{attribute addProperty BoxType "EL6201-0000-0017"}
{attribute addProperty Id "Slave_15A_DI0BIT10.125113Slave_15A_DI1BIT10.125114Slave_15A_DI2BIT10.125115Slave_15A_DI3BIT10.125116Slave_15B_DI0BIT10.125117Slave_15B_DI1BIT10.125118Slave_15B_DI2BIT10.125119Slave_15B_DI3BIT10.125120"}
{attribute addProperty CRC "3080739669"}
{attribute addProperty SizeInBites "8"}
{attribute addProperty SizeInBytes "1"}
TYPE Slave_15_Inputs_B7A05B55 :
STRUCT
	{attribute addProperty Name "Slave_15A_DI0"}
	Slave_15A_DI0 : BIT;
	{attribute addProperty Name "Slave_15A_DI1"}
	Slave_15A_DI1 : BIT;
	{attribute addProperty Name "Slave_15A_DI2"}
	Slave_15A_DI2 : BIT;
	{attribute addProperty Name "Slave_15A_DI3"}
	Slave_15A_DI3 : BIT;
	{attribute addProperty Name "Slave_15B_DI0"}
	Slave_15B_DI0 : BIT;
	{attribute addProperty Name "Slave_15B_DI1"}
	Slave_15B_DI1 : BIT;
	{attribute addProperty Name "Slave_15B_DI2"}
	Slave_15B_DI2 : BIT;
	{attribute addProperty Name "Slave_15B_DI3"}
	Slave_15B_DI3 : BIT;
END_STRUCT
END_TYPE

(* stored: Version 1.2.0.0, ProductVersion 3.1.4024.9
   DUT Slave_15_Inputs_B7A05B55: Id {9046cdec-39e5-4d50-b38f-2207dede95bc} *)
